// TIA Portal V21 export
TYPE "LBC_typeInterfaceCommands"
TITLE = LBC_typeInterfaceCommands
// Module related commands from external systems
   STRUCT
      refreshConfiguration : Bool;   // Copy global configuration parameters into module interface for external systems
      editConfiguration : Bool;   // Edit mode for configuration parameters in control system is active - copying into module interface is stopped
      saveConfiguration : Bool;   // Save configuration parameters from module interface into to global configuration parameters after change
      reset : Bool;   // Reinitialiazing the block
   END_STRUCT;
END_TYPE
